// TIA Portal V16 export
// export: Created 2024-05-10T06:46:45.5884281Z, ExportSetting WithDefaults, DisplayName Totally Integrated Automation Portal, DisplayVersion V16, DisplayName TIA Portal Version Control Interface, DisplayVersion V16, DisplayName TIA Portal Openness, DisplayVersion V16, DisplayName STEP 7 Professional, DisplayVersion V16, DisplayName STEP 7 Safety, DisplayVersion V16, DisplayName WinCC Professional, DisplayVersion V16
VAR_GLOBAL   // PLC tag table "106轴控制变量表"
   轴1定位1自动 AT %M2400.0 : Bool;
   轴1定位2自动 AT %M2400.1 : Bool;
   轴1定位3自动 AT %M2400.2 : Bool;
   轴1定位4自动 AT %M2400.3 : Bool;
   轴1xx1 AT %M2400.4 : Bool;
   轴1xx2 AT %M2400.5 : Bool;
   轴1xx3 AT %M2400.6 : Bool;
   轴1xx4 AT %M2400.7 : Bool;
   轴2定位1自动 AT %M2402.0 : Bool;
   轴2定位2自动 AT %M2402.1 : Bool;
   轴2定位3自动 AT %M2402.2 : Bool;
   轴2定位4自动 AT %M2402.3 : Bool;
   轴2xx1 AT %M2402.4 : Bool;
   轴2xx2 AT %M2402.5 : Bool;
   轴2xx3 AT %M2402.6 : Bool;
   轴2xx4 AT %M2402.7 : Bool;
   轴3定位1自动 AT %M2404.0 : Bool;
   轴3定位2自动 AT %M2404.1 : Bool;
   轴3定位3自动 AT %M2404.2 : Bool;
   轴3定位4自动 AT %M2404.3 : Bool;
   轴3xx1 AT %M2404.4 : Bool;
   轴3xx2 AT %M2404.5 : Bool;
   轴3xx3 AT %M2404.6 : Bool;
   轴3xx4 AT %M2404.7 : Bool;
   轴4定位1自动 AT %M2406.0 : Bool;
   轴4定位2自动 AT %M2406.1 : Bool;
   轴4定位3自动 AT %M2406.2 : Bool;
   轴4定位4自动 AT %M2406.3 : Bool;
   轴4xx1 AT %M2406.4 : Bool;
   轴4xx2 AT %M2406.5 : Bool;
   轴4xx3 AT %M2406.6 : Bool;
   轴4xx4 AT %M2406.7 : Bool;
   轴5定位1自动 AT %M2408.0 : Bool;
   轴5定位2自动 AT %M2408.1 : Bool;
   轴5定位3自动 AT %M2408.2 : Bool;
   轴5定位4自动 AT %M2408.3 : Bool;
   轴5xx1 AT %M2408.4 : Bool;
   轴5xx2 AT %M2408.5 : Bool;
   轴5xx3 AT %M2408.6 : Bool;
   轴5xx4 AT %M2408.7 : Bool;
   轴6定位1自动 AT %M2410.0 : Bool;
   轴6定位2自动 AT %M2410.1 : Bool;
   轴6定位3自动 AT %M2410.2 : Bool;
   轴6定位4自动 AT %M2410.3 : Bool;
   轴6xx1 AT %M2410.4 : Bool;
   轴6xx2 AT %M2410.5 : Bool;
   轴6xx3 AT %M2410.6 : Bool;
   轴6xx4 AT %M2410.7 : Bool;
   轴7定位1自动 AT %M2412.0 : Bool;
   轴7定位2自动 AT %M2412.1 : Bool;
   轴7定位3自动 AT %M2412.2 : Bool;
   轴7定位4自动 AT %M2412.3 : Bool;
   轴7xx1 AT %M2412.4 : Bool;
   轴7xx2 AT %M2412.5 : Bool;
   轴7xx3 AT %M2412.6 : Bool;
   轴7xx4 AT %M2412.7 : Bool;
   轴8定位1自动 AT %M2414.0 : Bool;
   轴8定位2自动 AT %M2414.1 : Bool;
   轴8定位3自动 AT %M2414.2 : Bool;
   轴8定位4自动 AT %M2414.3 : Bool;
   轴8xx1 AT %M2414.4 : Bool;
   轴8xx2 AT %M2414.5 : Bool;
   轴8xx3 AT %M2414.6 : Bool;
   轴8xx4 AT %M2414.7 : Bool;
   轴9定位1自动 AT %M2416.0 : Bool;
   轴9定位2自动 AT %M2416.1 : Bool;
   轴9定位3自动 AT %M2416.2 : Bool;
   轴9定位4自动 AT %M2416.3 : Bool;
   轴9xx1 AT %M2416.4 : Bool;
   轴9xx2 AT %M2416.5 : Bool;
   轴9xx3 AT %M2416.6 : Bool;
   轴9xx4 AT %M2416.7 : Bool;
   轴10定位1自动 AT %M2418.0 : Bool;
   轴10定位2自动 AT %M2418.1 : Bool;
   轴10定位3自动 AT %M2418.2 : Bool;
   轴10定位4自动 AT %M2418.3 : Bool;
   轴10xx1 AT %M2418.4 : Bool;
   轴10xx2 AT %M2418.5 : Bool;
   轴10xx3 AT %M2418.6 : Bool;
   轴10xx4 AT %M2418.7 : Bool;
   轴11定位1自动 AT %M2420.0 : Bool;
   轴11定位2自动 AT %M2420.1 : Bool;
   轴11定位3自动 AT %M2420.2 : Bool;
   轴11定位4自动 AT %M2420.3 : Bool;
   轴11xx1 AT %M2420.4 : Bool;
   轴11xx2 AT %M2420.5 : Bool;
   轴11xx3 AT %M2420.6 : Bool;
   轴11xx4 AT %M2420.7 : Bool;
   轴12定位1自动 AT %M2422.0 : Bool;
   轴12定位2自动 AT %M2422.1 : Bool;
   轴12定位3自动 AT %M2422.2 : Bool;
   轴12定位4自动 AT %M2422.3 : Bool;
   轴12xx1 AT %M2422.4 : Bool;
   轴12xx2 AT %M2422.5 : Bool;
   轴12xx3 AT %M2422.6 : Bool;
   轴12xx4 AT %M2422.7 : Bool;
   轴13定位1自动 AT %M2424.0 : Bool;
   轴13定位2自动 AT %M2424.1 : Bool;
   轴13定位3自动 AT %M2424.2 : Bool;
   轴13定位4自动 AT %M2424.3 : Bool;
   轴13xx1 AT %M2424.4 : Bool;
   轴13xx2 AT %M2424.5 : Bool;
   轴13xx3 AT %M2424.6 : Bool;
   轴13xx4 AT %M2424.7 : Bool;
   轴14定位1自动 AT %M2426.0 : Bool;
   轴14定位2自动 AT %M2426.1 : Bool;
   轴14定位3自动 AT %M2426.2 : Bool;
   轴14定位4自动 AT %M2426.3 : Bool;
   轴14xx1 AT %M2426.4 : Bool;
   轴14xx2 AT %M2426.5 : Bool;
   轴14xx3 AT %M2426.6 : Bool;
   轴14xx4 AT %M2426.7 : Bool;
   轴15定位1自动 AT %M2428.0 : Bool;
   轴15定位2自动 AT %M2428.1 : Bool;
   轴15定位3自动 AT %M2428.2 : Bool;
   轴15定位4自动 AT %M2428.3 : Bool;
   轴15xx1 AT %M2428.4 : Bool;
   轴15xx2 AT %M2428.5 : Bool;
   轴15xx3 AT %M2428.6 : Bool;
   轴15xx4 AT %M2428.7 : Bool;
   轴16定位1自动 AT %M2430.0 : Bool;
   轴16定位2自动 AT %M2430.1 : Bool;
   轴16定位3自动 AT %M2430.2 : Bool;
   轴16定位4自动 AT %M2430.3 : Bool;
   轴16xx1 AT %M2430.4 : Bool;
   轴16xx2 AT %M2430.5 : Bool;
   轴16xx3 AT %M2430.6 : Bool;
   轴16xx4 AT %M2430.7 : Bool;
   XXXXXX1 AT %M2432.0 : Bool;
   轴1定位1手动 AT %M1400.0 : Bool;
   轴1定位2手动 AT %M1400.1 : Bool;
   轴1定位3手动 AT %M1400.2 : Bool;
   轴1定位4手动 AT %M1400.3 : Bool;
   轴1xx1手动 AT %M1400.4 : Bool;
   轴1xx2手动 AT %M1400.5 : Bool;
   轴1xx3手动 AT %M1400.6 : Bool;
   轴1xx4手动 AT %M1400.7 : Bool;
   轴1使能 AT %M1401.0 : Bool;
   轴1回零 AT %M1401.1 : Bool;
   "轴1点动+" AT %M1401.2 : Bool;
   "轴1点动-" AT %M1401.3 : Bool;
   轴1自由定位 AT %M1401.4 : Bool;
   轴1就绪 AT %M1401.5 : Bool;
   轴1原点 AT %M1401.6 : Bool;
   轴1到达 AT %M1401.7 : Bool;
   轴2定位1手动 AT %M1402.0 : Bool;
   轴2定位2手动 AT %M1402.1 : Bool;
   轴2定位3手动 AT %M1402.2 : Bool;
   轴2定位4手动 AT %M1402.3 : Bool;
   轴2xx1手动 AT %M1402.4 : Bool;
   轴2xx2手动 AT %M1402.5 : Bool;
   轴2xx3手动 AT %M1402.6 : Bool;
   轴2xx4手动 AT %M1402.7 : Bool;
   轴2使能 AT %M1403.0 : Bool;
   轴2回零 AT %M1403.1 : Bool;
   "轴2点动+" AT %M1403.2 : Bool;
   "轴2点动-" AT %M1403.3 : Bool;
   轴2自由定位 AT %M1403.4 : Bool;
   轴2就绪 AT %M1403.5 : Bool;
   轴2原点 AT %M1403.6 : Bool;
   轴2到达 AT %M1403.7 : Bool;
   轴3定位1手动 AT %M1404.0 : Bool;
   轴3定位2手动 AT %M1404.1 : Bool;
   轴3定位3手动 AT %M1404.2 : Bool;
   轴3定位4手动 AT %M1404.3 : Bool;
   轴3xx1手动 AT %M1404.4 : Bool;
   轴3xx2手动 AT %M1404.5 : Bool;
   轴3xx3手动 AT %M1404.6 : Bool;
   轴3xx4手动 AT %M1404.7 : Bool;
   轴3使能 AT %M1405.0 : Bool;
   轴3回零 AT %M1405.1 : Bool;
   "轴3点动+" AT %M1405.2 : Bool;
   "轴3点动-" AT %M1405.3 : Bool;
   轴3自由定位 AT %M1405.4 : Bool;
   轴3就绪 AT %M1405.5 : Bool;
   轴3原点 AT %M1405.6 : Bool;
   轴3到达 AT %M1405.7 : Bool;
   轴4定位1手动 AT %M1406.0 : Bool;
   轴4定位2手动 AT %M1406.1 : Bool;
   轴4定位3手动 AT %M1406.2 : Bool;
   轴4自由定位 AT %M1407.4 : Bool;
   轴4xx1手动 AT %M1406.4 : Bool;
   轴4xx2手动 AT %M1406.5 : Bool;
   轴4xx3手动 AT %M1406.6 : Bool;
   轴4xx4手动 AT %M1406.7 : Bool;
   轴4使能 AT %M1407.0 : Bool;
   轴4回零 AT %M1407.1 : Bool;
   "轴4点动+" AT %M1407.2 : Bool;
   "轴4点动-" AT %M1407.3 : Bool;
   轴4就绪 AT %M1407.5 : Bool;
   轴4原点 AT %M1407.6 : Bool;
   轴4到达 AT %M1407.7 : Bool;
   轴5定位1手动 AT %M1408.0 : Bool;
   轴5定位2手动 AT %M1408.1 : Bool;
   轴5定位3手动 AT %M1408.2 : Bool;
   轴5定位4手动 AT %M1408.3 : Bool;
   轴5xx1手动 AT %M1408.4 : Bool;
   轴5xx2手动 AT %M1408.5 : Bool;
   轴5xx3手动 AT %M1408.6 : Bool;
   轴5xx4手动 AT %M1408.7 : Bool;
   轴5使能 AT %M1409.0 : Bool;
   轴5回零 AT %M1409.1 : Bool;
   "轴5点动+" AT %M1409.2 : Bool;
   "轴5点动-" AT %M1409.3 : Bool;
   轴5自由定位 AT %M1409.4 : Bool;
   轴5就绪 AT %M1409.5 : Bool;
   轴5原点 AT %M1409.6 : Bool;
   轴5到达 AT %M1409.7 : Bool;
   轴6定位1手动 AT %M1410.0 : Bool;
   轴6定位2手动 AT %M1410.1 : Bool;
   轴6定位3手动 AT %M1410.2 : Bool;
   轴6定位4手动 AT %M1410.3 : Bool;
   轴6xx1手动 AT %M1410.4 : Bool;
   轴6xx2手动 AT %M1410.5 : Bool;
   轴6xx3手动 AT %M1410.6 : Bool;
   轴6xx4手动 AT %M1410.7 : Bool;
   轴6使能 AT %M1411.0 : Bool;
   轴6回零 AT %M1411.1 : Bool;
   "轴6点动+" AT %M1411.2 : Bool;
   "轴6点动-" AT %M1411.3 : Bool;
   轴6自由定位 AT %M1411.4 : Bool;
   轴6就绪 AT %M1411.5 : Bool;
   轴6原点 AT %M1411.6 : Bool;
   轴6到达 AT %M1411.7 : Bool;
   轴7定位1手动 AT %M1412.0 : Bool;
   轴7定位2手动 AT %M1412.1 : Bool;
   轴7定位3手动 AT %M1412.2 : Bool;
   轴7定位4手动 AT %M1412.3 : Bool;
   轴7xx1手动 AT %M1412.4 : Bool;
   轴7xx2手动 AT %M1412.5 : Bool;
   轴7xx3手动 AT %M1412.6 : Bool;
   轴7xx4手动 AT %M1412.7 : Bool;
   轴7使能 AT %M1413.0 : Bool;
   轴7回零 AT %M1413.1 : Bool;
   "轴7点动+" AT %M1413.2 : Bool;
   "轴7点动-" AT %M1413.3 : Bool;
   轴7自由定位 AT %M1413.4 : Bool;
   轴7就绪 AT %M1413.5 : Bool;
   轴7原点 AT %M1413.6 : Bool;
   轴7到达 AT %M1413.7 : Bool;
   轴8定位1手动 AT %M1414.0 : Bool;
   轴8定位2手动 AT %M1414.1 : Bool;
   轴8定位3手动 AT %M1414.2 : Bool;
   轴8定位4手动 AT %M1414.3 : Bool;
   轴8xx1手动 AT %M1414.4 : Bool;
   轴8xx2手动 AT %M1414.5 : Bool;
   轴8xx3手动 AT %M1414.6 : Bool;
   轴8xx4手动 AT %M1414.7 : Bool;
   轴8使能 AT %M1415.0 : Bool;
   轴8回零 AT %M1415.1 : Bool;
   "轴8点动+" AT %M1415.2 : Bool;
   "轴8点动-" AT %M1415.3 : Bool;
   轴8自由定位 AT %M1415.4 : Bool;
   轴8就绪 AT %M1415.5 : Bool;
   轴8原点 AT %M1415.6 : Bool;
   轴8到达 AT %M1415.7 : Bool;
   轴9定位1手动 AT %M1416.0 : Bool;
   轴9定位2手动 AT %M1416.1 : Bool;
   轴9定位3手动 AT %M1416.2 : Bool;
   轴9定位4手动 AT %M1416.3 : Bool;
   轴9xx1手动 AT %M1416.4 : Bool;
   轴9xx2手动 AT %M1416.5 : Bool;
   轴9xx3手动 AT %M1416.6 : Bool;
   轴9xx4手动 AT %M1416.7 : Bool;
   轴9使能 AT %M1417.0 : Bool;
   轴9回零 AT %M1417.1 : Bool;
   "轴9点动+" AT %M1417.2 : Bool;
   "轴9点动-" AT %M1417.3 : Bool;
   轴9自由定位 AT %M1417.4 : Bool;
   轴9就绪 AT %M1417.5 : Bool;
   轴9原点 AT %M1417.6 : Bool;
   轴9到达 AT %M1417.7 : Bool;
   轴10定位1手动 AT %M1418.0 : Bool;
   轴10定位2手动 AT %M1418.1 : Bool;
   轴10定位3手动 AT %M1418.2 : Bool;
   轴10定位4手动 AT %M1418.3 : Bool;
   轴10xx1手动 AT %M1418.4 : Bool;
   轴10xx2手动 AT %M1418.5 : Bool;
   轴10xx3手动 AT %M1418.6 : Bool;
   轴10xx4手动 AT %M1418.7 : Bool;
   轴10使能 AT %M1419.0 : Bool;
   轴10回零 AT %M1419.1 : Bool;
   "轴10点动+" AT %M1419.2 : Bool;
   "轴10点动-" AT %M1419.3 : Bool;
   轴10自由定位 AT %M1419.4 : Bool;
   轴10就绪 AT %M1419.5 : Bool;
   轴10原点 AT %M1419.6 : Bool;
   轴10到达 AT %M1419.7 : Bool;
   轴11定位1手动 AT %M1420.0 : Bool;
   轴11定位2手动 AT %M1420.1 : Bool;
   轴11定位3手动 AT %M1420.2 : Bool;
   轴11定位4手动 AT %M1420.3 : Bool;
   轴11xx1手动 AT %M1420.4 : Bool;
   轴11xx2手动 AT %M1420.5 : Bool;
   轴11xx3手动 AT %M1420.6 : Bool;
   轴11xx4手动 AT %M1420.7 : Bool;
   轴11使能 AT %M1421.0 : Bool;
   轴11回零 AT %M1421.1 : Bool;
   "轴11点动+" AT %M1421.2 : Bool;
   "轴11点动-" AT %M1421.3 : Bool;
   轴11自由定位 AT %M1421.4 : Bool;
   轴11就绪 AT %M1421.5 : Bool;
   轴11原点 AT %M1421.6 : Bool;
   轴11到达 AT %M1421.7 : Bool;
   轴12定位1手动 AT %M1422.0 : Bool;
   轴12定位2手动 AT %M1422.1 : Bool;
   轴12定位3手动 AT %M1422.2 : Bool;
   轴12定位4手动 AT %M1422.3 : Bool;
   轴12xx1手动 AT %M1422.4 : Bool;
   轴12xx2手动 AT %M1422.5 : Bool;
   轴12xx3手动 AT %M1422.6 : Bool;
   轴12xx4手动 AT %M1422.7 : Bool;
   轴12使能 AT %M1423.0 : Bool;
   轴12回零 AT %M1423.1 : Bool;
   "轴12点动+" AT %M1423.2 : Bool;
   "轴12点动-" AT %M1423.3 : Bool;
   轴12自由定位 AT %M1423.4 : Bool;
   轴12就绪 AT %M1423.5 : Bool;
   轴12原点 AT %M1423.6 : Bool;
   轴12到达 AT %M1423.7 : Bool;
   轴13定位1手动 AT %M1424.0 : Bool;
   轴13定位2手动 AT %M1424.1 : Bool;
   轴13定位3手动 AT %M1424.2 : Bool;
   轴13定位4手动 AT %M1424.3 : Bool;
   轴13xx1手动 AT %M1424.4 : Bool;
   轴13xx2手动 AT %M1424.5 : Bool;
   轴13xx3手动 AT %M1424.6 : Bool;
   轴13xx4手动 AT %M1424.7 : Bool;
   轴13使能 AT %M1425.0 : Bool;
   轴13回零 AT %M1425.1 : Bool;
   "轴13点动+" AT %M1425.2 : Bool;
   "轴13点动-" AT %M1425.3 : Bool;
   轴13自由定位 AT %M1425.4 : Bool;
   轴13就绪 AT %M1425.5 : Bool;
   轴13原点 AT %M1425.6 : Bool;
   轴13到达 AT %M1425.7 : Bool;
   轴14定位1手动 AT %M1426.0 : Bool;
   轴14定位2手动 AT %M1426.1 : Bool;
   轴14定位3手动 AT %M1426.2 : Bool;
   轴14定位4手动 AT %M1426.3 : Bool;
   轴14xx1手动 AT %M1426.4 : Bool;
   轴14xx2手动 AT %M1426.5 : Bool;
   轴14xx3手动 AT %M1426.6 : Bool;
   轴14xx4手动 AT %M1426.7 : Bool;
   轴14使能 AT %M1427.0 : Bool;
   轴14回零 AT %M1427.1 : Bool;
   "轴14点动+" AT %M1427.2 : Bool;
   "轴14点动-" AT %M1427.3 : Bool;
   轴14自由定位 AT %M1427.4 : Bool;
   轴14就绪 AT %M1427.5 : Bool;
   轴14原点 AT %M1427.6 : Bool;
   轴14到达 AT %M1427.7 : Bool;
   轴15定位1手动 AT %M1428.0 : Bool;
   轴15定位2手动 AT %M1428.1 : Bool;
   轴15定位3手动 AT %M1428.2 : Bool;
   轴15定位4手动 AT %M1428.3 : Bool;
   轴15xx1手动 AT %M1428.4 : Bool;
   轴15xx2手动 AT %M1428.5 : Bool;
   轴15xx3手动 AT %M1428.6 : Bool;
   轴15xx4手动 AT %M1428.7 : Bool;
   轴15使能 AT %M1429.0 : Bool;
   轴15回零 AT %M1429.1 : Bool;
   "轴15点动+" AT %M1429.2 : Bool;
   "轴15点动-" AT %M1429.3 : Bool;
   轴15自由定位 AT %M1429.4 : Bool;
   轴15就绪 AT %M1429.5 : Bool;
   轴15原点 AT %M1429.6 : Bool;
   轴15到达 AT %M1429.7 : Bool;
   轴16定位1手动 AT %M1430.0 : Bool;
   轴16定位2手动 AT %M1430.1 : Bool;
   轴16定位3手动 AT %M1430.2 : Bool;
   轴16定位4手动 AT %M1430.3 : Bool;
   轴16xx1手动 AT %M1430.4 : Bool;
   轴16xx2手动 AT %M1430.5 : Bool;
   轴16xx3手动 AT %M1430.6 : Bool;
   轴16xx4手动 AT %M1430.7 : Bool;
   轴16使能 AT %M1431.0 : Bool;
   轴16回零 AT %M1431.1 : Bool;
   "轴16点动+" AT %M1431.2 : Bool;
   "轴16点动-" AT %M1431.3 : Bool;
   轴16自由定位 AT %M1431.4 : Bool;
   轴16就绪 AT %M1431.5 : Bool;
   轴16原点 AT %M1431.6 : Bool;
   轴16到达 AT %M1431.7 : Bool;
   XXXXXX2 AT %M1432.0 : Bool;
   轴1定位1到位 AT %M3400.0 : Bool;
   轴1定位2到位 AT %M3400.1 : Bool;
   轴1定位3到位 AT %M3400.2 : Bool;
   轴1定位4到位 AT %M3400.3 : Bool;
   轴2定位1到位 AT %M3401.0 : Bool;
   轴2定位2到位 AT %M3401.1 : Bool;
   轴2定位3到位 AT %M3401.2 : Bool;
   轴2定位4到位 AT %M3401.3 : Bool;
   轴3定位1到位 AT %M3402.0 : Bool;
   轴3定位2到位 AT %M3402.1 : Bool;
   轴3定位3到位 AT %M3402.2 : Bool;
   轴3定位4到位 AT %M3402.3 : Bool;
   轴4定位1到位 AT %M3403.0 : Bool;
   轴4定位2到位 AT %M3403.1 : Bool;
   轴4定位3到位 AT %M3403.2 : Bool;
   轴4定位4到位 AT %M3403.3 : Bool;
   轴5定位1到位 AT %M3404.0 : Bool;
   轴5定位2到位 AT %M3404.1 : Bool;
   轴5定位3到位 AT %M3404.2 : Bool;
   轴5定位4到位 AT %M3404.3 : Bool;
   轴6定位1到位 AT %M3405.0 : Bool;
   轴6定位2到位 AT %M3405.1 : Bool;
   轴6定位3到位 AT %M3405.2 : Bool;
   轴6定位4到位 AT %M3405.3 : Bool;
   轴7定位1到位 AT %M3406.0 : Bool;
   轴7定位2到位 AT %M3406.1 : Bool;
   轴7定位3到位 AT %M3406.2 : Bool;
   轴7定位4到位 AT %M3406.3 : Bool;
   轴8定位1到位 AT %M3407.0 : Bool;
   轴8定位2到位 AT %M3407.1 : Bool;
   轴8定位3到位 AT %M3407.2 : Bool;
   轴8定位4到位 AT %M3407.3 : Bool;
   轴9定位1到位 AT %M3408.0 : Bool;
   轴9定位2到位 AT %M3408.1 : Bool;
   轴9定位3到位 AT %M3408.2 : Bool;
   轴9定位4到位 AT %M3408.3 : Bool;
   轴10定位1到位 AT %M3409.0 : Bool;
   轴10定位2到位 AT %M3409.1 : Bool;
   轴10定位3到位 AT %M3409.2 : Bool;
   轴10定位4到位 AT %M3409.3 : Bool;
   轴11定位1到位 AT %M3410.0 : Bool;
   轴11定位2到位 AT %M3410.1 : Bool;
   轴11定位3到位 AT %M3410.2 : Bool;
   轴11定位4到位 AT %M3410.3 : Bool;
   轴12定位1到位 AT %M3411.0 : Bool;
   轴12定位2到位 AT %M3411.1 : Bool;
   轴12定位3到位 AT %M3411.2 : Bool;
   轴12定位4到位 AT %M3411.3 : Bool;
   轴13定位1到位 AT %M3412.0 : Bool;
   轴13定位2到位 AT %M3412.1 : Bool;
   轴13定位3到位 AT %M3412.2 : Bool;
   轴13定位4到位 AT %M3412.3 : Bool;
   轴14定位1到位 AT %M3413.0 : Bool;
   轴14定位2到位 AT %M3413.1 : Bool;
   轴14定位3到位 AT %M3413.2 : Bool;
   轴14定位4到位 AT %M3413.3 : Bool;
   轴15定位1到位 AT %M3414.0 : Bool;
   轴15定位2到位 AT %M3414.1 : Bool;
   轴15定位3到位 AT %M3414.2 : Bool;
   轴15定位4到位 AT %M3414.3 : Bool;
   轴16定位1到位 AT %M3415.0 : Bool;
   轴16定位2到位 AT %M3415.1 : Bool;
   轴16定位3到位 AT %M3415.2 : Bool;
   轴16定位4到位 AT %M3415.3 : Bool;
   XXXXXX3 AT %M3416.0 : Bool;
   轴1回零高速 AT %MD1500 : DInt;
   轴1回零低速 AT %MD1504 : DInt;
   轴1点动速度 AT %MD1508 : DInt;
   轴1最高速度 AT %MD1512 : DInt;
   轴1自由定位值 AT %MD1516 : DInt;
   轴2回零高速 AT %MD1520 : DInt;
   轴2回零低速 AT %MD1524 : DInt;
   轴2点动速度 AT %MD1528 : DInt;
   轴2最高速度 AT %MD1532 : DInt;
   轴2自由定位值 AT %MD1536 : DInt;
   轴3回零高速 AT %MD1540 : DInt;
   轴3回零低速 AT %MD1544 : DInt;
   轴3点动速度 AT %MD1548 : DInt;
   轴3最高速度 AT %MD1552 : DInt;
   轴3自由定位值 AT %MD1556 : DInt;
   轴4回零高速 AT %MD1560 : DInt;
   轴4回零低速 AT %MD1564 : DInt;
   轴4点动速度 AT %MD1568 : DInt;
   轴4最高速度 AT %MD1572 : DInt;
   轴4自由定位值 AT %MD1576 : DInt;
   轴5回零高速 AT %MD1580 : DInt;
   轴5回零低速 AT %MD1584 : DInt;
   轴5点动速度 AT %MD1588 : DInt;
   轴5最高速度 AT %MD1592 : DInt;
   轴5自由定位值 AT %MD1596 : DInt;
   轴6回零高速 AT %MD1600 : DInt;
   轴6回零低速 AT %MD1604 : DInt;
   轴6点动速度 AT %MD1608 : DInt;
   轴6最高速度 AT %MD1612 : DInt;
   轴6自由定位值 AT %MD1616 : DInt;
   轴7回零高速 AT %MD1620 : DInt;
   轴7回零低速 AT %MD1624 : DInt;
   轴7点动速度 AT %MD1628 : DInt;
   轴7最高速度 AT %MD1632 : DInt;
   轴7自由定位值 AT %MD1636 : DInt;
   轴8回零高速 AT %MD1640 : DInt;
   轴8回零低速 AT %MD1644 : DInt;
   轴8点动速度 AT %MD1648 : DInt;
   轴8最高速度 AT %MD1652 : DInt;
   轴8自由定位值 AT %MD1656 : DInt;
   轴9回零高速 AT %MD1660 : DInt;
   轴9回零低速 AT %MD1664 : DInt;
   轴9点动速度 AT %MD1668 : DInt;
   轴9最高速度 AT %MD1672 : DInt;
   轴9自由定位值 AT %MD1676 : DInt;
   轴10回零高速 AT %MD1680 : DInt;
   轴10回零低速 AT %MD1684 : DInt;
   轴10点动速度 AT %MD1688 : DInt;
   轴10最高速度 AT %MD1692 : DInt;
   轴10自由定位值 AT %MD1696 : DInt;
   轴11回零高速 AT %MD1700 : DInt;
   轴11回零低速 AT %MD1704 : DInt;
   轴11点动速度 AT %MD1708 : DInt;
   轴11最高速度 AT %MD1712 : DInt;
   轴11自由定位值 AT %MD1716 : DInt;
   轴12回零高速 AT %MD1720 : DInt;
   轴12回零低速 AT %MD1724 : DInt;
   轴12点动速度 AT %MD1728 : DInt;
   轴12最高速度 AT %MD1732 : DInt;
   轴12自由定位值 AT %MD1736 : DInt;
   轴13回零高速 AT %MD1740 : DInt;
   轴13回零低速 AT %MD1744 : DInt;
   轴13点动速度 AT %MD1748 : DInt;
   轴13最高速度 AT %MD1752 : DInt;
   轴13自由定位值 AT %MD1756 : DInt;
   轴14回零高速 AT %MD1760 : DInt;
   轴14回零低速 AT %MD1764 : DInt;
   轴14点动速度 AT %MD1768 : DInt;
   轴14最高速度 AT %MD1772 : DInt;
   轴14自由定位值 AT %MD1776 : DInt;
   轴15回零高速 AT %MD1780 : DInt;
   轴15回零低速 AT %MD1784 : DInt;
   轴15点动速度 AT %MD1788 : DInt;
   轴15最高速度 AT %MD1792 : DInt;
   轴15自由定位值 AT %MD1796 : DInt;
   轴16回零高速 AT %MD1800 : DInt;
   轴16回零低速 AT %MD1804 : DInt;
   轴16点动速度 AT %MD1808 : DInt;
   轴16最高速度 AT %MD1812 : DInt;
   轴16自由定位值 AT %MD1816 : DInt;
   XXXXXX4 AT %MW1920 : Int;
   轴1位置1 AT %MD2500 : DInt;
   轴1位置2 AT %MD2504 : DInt;
   轴1位置3 AT %MD2508 : DInt;
   轴1位置4 AT %MD2512 : DInt;
   轴2位置1 AT %MD2520 : DInt;
   轴2位置2 AT %MD2524 : DInt;
   轴2位置3 AT %MD2528 : DInt;
   轴2位置4 AT %MD2532 : DInt;
   轴3位置1 AT %MD2540 : DInt;
   轴3位置2 AT %MD2544 : DInt;
   轴3位置3 AT %MD2548 : DInt;
   轴3位置4 AT %MD2552 : DInt;
   轴4位置1 AT %MD2560 : DInt;
   轴4位置2 AT %MD2564 : DInt;
   轴4位置3 AT %MD2568 : DInt;
   轴4位置4 AT %MD2572 : DInt;
   轴5位置1 AT %MD2580 : DInt;
   轴5位置2 AT %MD2584 : DInt;
   轴5位置3 AT %MD2588 : DInt;
   轴5位置4 AT %MD2592 : DInt;
   轴6位置1 AT %MD2600 : DInt;
   轴6位置2 AT %MD2604 : DInt;
   轴6位置3 AT %MD2608 : DInt;
   轴6位置4 AT %MD2612 : DInt;
   轴7位置1 AT %MD2620 : DInt;
   轴7位置2 AT %MD2624 : DInt;
   轴7位置3 AT %MD2628 : DInt;
   轴7位置4 AT %MD2632 : DInt;
   轴8位置1 AT %MD2640 : DInt;
   轴8位置2 AT %MD2644 : DInt;
   轴8位置3 AT %MD2648 : DInt;
   轴8位置4 AT %MD2652 : DInt;
   轴9位置1 AT %MD2660 : DInt;
   轴9位置2 AT %MD2664 : DInt;
   轴9位置3 AT %MD2668 : DInt;
   轴9位置4 AT %MD2672 : DInt;
   轴10位置1 AT %MD2680 : DInt;
   轴10位置2 AT %MD2684 : DInt;
   轴10位置3 AT %MD2688 : DInt;
   轴10位置4 AT %MD2692 : DInt;
   轴11位置1 AT %MD2700 : DInt;
   轴11位置2 AT %MD2704 : DInt;
   轴11位置3 AT %MD2708 : DInt;
   轴11位置4 AT %MD2712 : DInt;
   轴12位置1 AT %MD2720 : DInt;
   轴12位置2 AT %MD2724 : DInt;
   轴12位置3 AT %MD2728 : DInt;
   轴12位置4 AT %MD2732 : DInt;
   轴13位置1 AT %MD2740 : DInt;
   轴13位置2 AT %MD2744 : DInt;
   轴13位置3 AT %MD2748 : DInt;
   轴13位置4 AT %MD2752 : DInt;
   轴14位置1 AT %MD2760 : DInt;
   轴14位置2 AT %MD2764 : DInt;
   轴14位置3 AT %MD2768 : DInt;
   轴14位置4 AT %MD2772 : DInt;
   轴15位置1 AT %MD2780 : DInt;
   轴15位置2 AT %MD2784 : DInt;
   轴15位置3 AT %MD2788 : DInt;
   轴15位置4 AT %MD2792 : DInt;
   轴16位置1 AT %MD2800 : DInt;
   轴16位置2 AT %MD2804 : DInt;
   轴16位置3 AT %MD2808 : DInt;
   轴16位置4 AT %MD2812 : DInt;
   XXXXXX5 AT %MW2820 : Int;
   轴1速度1 AT %MW3500 : Int;
   轴1速度2 AT %MW3504 : Int;
   轴1速度3 AT %MW3508 : Int;
   轴1速度4 AT %MW3512 : Int;
   轴2速度1 AT %MW3520 : Int;
   轴2速度2 AT %MW3524 : Int;
   轴2速度3 AT %MW3528 : Int;
   轴2速度4 AT %MW3532 : Int;
   轴3速度1 AT %MW3540 : Int;
   轴3速度2 AT %MW3544 : Int;
   轴3速度3 AT %MW3548 : Int;
   轴3速度4 AT %MW3552 : Int;
   轴4速度1 AT %MW3560 : Int;
   轴4速度2 AT %MW3564 : Int;
   轴4速度3 AT %MW3568 : Int;
   轴4速度4 AT %MW3572 : Int;
   轴5速度1 AT %MW3580 : Int;
   轴5速度2 AT %MW3584 : Int;
   轴5速度3 AT %MW3588 : Int;
   轴5速度4 AT %MW3592 : Int;
   轴6速度1 AT %MW3600 : Int;
   轴6速度2 AT %MW3604 : Int;
   轴6速度3 AT %MW3608 : Int;
   轴6速度4 AT %MW3612 : Int;
   轴7速度1 AT %MW3620 : Int;
   轴7速度2 AT %MW3624 : Int;
   轴7速度3 AT %MW3628 : Int;
   轴7速度4 AT %MW3632 : Int;
   轴8速度1 AT %MW3640 : Int;
   轴8速度2 AT %MW3644 : Int;
   轴8速度3 AT %MW3648 : Int;
   轴8速度4 AT %MW3652 : Int;
   轴9速度1 AT %MW3660 : Int;
   轴9速度2 AT %MW3664 : Int;
   轴9速度3 AT %MW3668 : Int;
   轴9速度4 AT %MW3672 : Int;
   轴10速度1 AT %MW3680 : Int;
   轴10速度2 AT %MW3684 : Int;
   轴10速度3 AT %MW3688 : Int;
   轴10速度4 AT %MW3692 : Int;
   轴11速度1 AT %MW3700 : Int;
   轴11速度2 AT %MW3704 : Int;
   轴11速度3 AT %MW3708 : Int;
   轴11速度4 AT %MW3712 : Int;
   轴12速度1 AT %MW3720 : Int;
   轴12速度2 AT %MW3724 : Int;
   轴12速度3 AT %MW3728 : Int;
   轴12速度4 AT %MW3732 : Int;
   轴13速度1 AT %MW3740 : Int;
   轴13速度2 AT %MW3744 : Int;
   轴13速度3 AT %MW3748 : Int;
   轴13速度4 AT %MW3752 : Int;
   轴14速度1 AT %MW3760 : Int;
   轴14速度2 AT %MW3764 : Int;
   轴14速度3 AT %MW3768 : Int;
   轴14速度4 AT %MW3772 : Int;
   轴15速度1 AT %MW3780 : Int;
   轴15速度2 AT %MW3784 : Int;
   轴15速度3 AT %MW3788 : Int;
   轴15速度4 AT %MW3792 : Int;
   轴16速度1 AT %MW3800 : Int;
   轴16速度2 AT %MW3804 : Int;
   轴16速度3 AT %MW3808 : Int;
   轴16速度4 AT %MW3812 : Int;
   XXXXXX6 AT %MW3820 : Int;
   轴01目标位置 AT %MD4500 : DInt;
   轴02目标位置 AT %MD4504 : DInt;
   轴03目标位置 AT %MD4508 : DInt;
   轴04目标位置 AT %MD4512 : DInt;
   轴05目标位置 AT %MD4516 : DInt;
   轴06目标位置 AT %MD4520 : DInt;
   轴07目标位置 AT %MD4524 : DInt;
   轴08目标位置 AT %MD4528 : DInt;
   轴09目标位置 AT %MD4532 : DInt;
   轴10目标位置 AT %MD4536 : DInt;
   轴11目标位置 AT %MD4540 : DInt;
   轴12目标位置 AT %MD4544 : DInt;
   轴13目标位置 AT %MD4548 : DInt;
   轴14目标位置 AT %MD4552 : DInt;
   轴15目标位置 AT %MD4556 : DInt;
   轴16目标位置 AT %MD4560 : DInt;
   XXXXXX7 AT %MD4564 : DInt;
   轴01目标速度 AT %MD4600 : DInt;
   轴02目标速度 AT %MD4604 : DInt;
   轴03目标速度 AT %MD4608 : DInt;
   轴04目标速度 AT %MD4612 : DInt;
   轴05目标速度 AT %MD4616 : DInt;
   轴06目标速度 AT %MD4620 : DInt;
   轴07目标速度 AT %MD4624 : DInt;
   轴08目标速度 AT %MD4628 : DInt;
   轴09目标速度 AT %MD4632 : DInt;
   轴10目标速度 AT %MD4636 : DInt;
   轴11目标速度 AT %MD4640 : DInt;
   轴12目标速度 AT %MD4644 : DInt;
   轴13目标速度 AT %MD4648 : DInt;
   轴14目标速度 AT %MD4652 : DInt;
   轴15目标速度 AT %MD4656 : DInt;
   轴16目标速度 AT %MD4660 : DInt;
   XXXXXX8 AT %MD4664 : DInt;
   轴01当前位置 AT %MD4700 : DInt;
   轴02当前位置 AT %MD4704 : DInt;
   轴03当前位置 AT %MD4708 : DInt;
   轴04当前位置 AT %MD4712 : DInt;
   轴05当前位置 AT %MD4716 : DInt;
   轴06当前位置 AT %MD4720 : DInt;
   轴07当前位置 AT %MD4724 : DInt;
   轴08当前位置 AT %MD4728 : DInt;
   轴09当前位置 AT %MD4732 : DInt;
   轴10当前位置 AT %MD4736 : DInt;
   轴11当前位置 AT %MD4740 : DInt;
   轴12当前位置 AT %MD4744 : DInt;
   轴13当前位置 AT %MD4748 : DInt;
   轴14当前位置 AT %MD4752 : DInt;
   轴15当前位置 AT %MD4756 : DInt;
   轴16当前位置 AT %MD4760 : DInt;
   XXXXXX9 AT %MD4764 : DInt;
   轴01当前速度 AT %MD4800 : DInt;
   轴02当前速度 AT %MD4804 : DInt;
   轴03当前速度 AT %MD4808 : DInt;
   轴04当前速度 AT %MD4812 : DInt;
   轴05当前速度 AT %MD4816 : DInt;
   轴06当前速度 AT %MD4820 : DInt;
   轴07当前速度 AT %MD4824 : DInt;
   轴08当前速度 AT %MD4828 : DInt;
   轴09当前速度 AT %MD4832 : DInt;
   轴10当前速度 AT %MD4836 : DInt;
   轴11当前速度 AT %MD4840 : DInt;
   轴12当前速度 AT %MD4844 : DInt;
   轴13当前速度 AT %MD4848 : DInt;
   轴14当前速度 AT %MD4852 : DInt;
   轴15当前速度 AT %MD4856 : DInt;
   轴16当前速度 AT %MD4860 : DInt;
   XXXXXX10 AT %MD4864 : DInt;
   轴1报警码 AT %MW4900 : Word;
   轴2报警码 AT %MW4901 : Word;
   轴3报警码 AT %MW4902 : Word;
   轴4报警码 AT %MW4903 : Word;
   轴5报警码 AT %MW4904 : Word;
   轴6报警码 AT %MW4905 : Word;
   轴7报警码 AT %MW4906 : Word;
   轴8报警码 AT %MW4907 : Word;
   轴9报警码 AT %MW4908 : Word;
   轴10报警码 AT %MW4909 : Word;
   轴11报警码 AT %MW4910 : Word;
   轴12报警码 AT %MW4911 : Word;
   轴13报警码 AT %MW4912 : Word;
   轴14报警码 AT %MW4913 : Word;
   轴15报警码 AT %MW4914 : Word;
   轴16报警码 AT %MW4915 : Word;
   XXXXXX11 AT %MW4916 : Word;
   轴1错误码 AT %MW4920 : Word;
   轴2错误码 AT %MW4921 : Word;
   轴3错误码 AT %MW4922 : Word;
   轴4错误码 AT %MW4923 : Word;
   轴5错误码 AT %MW4924 : Word;
   轴6错误码 AT %MW4925 : Word;
   轴7错误码 AT %MW4926 : Word;
   轴8错误码 AT %MW4927 : Word;
   轴9错误码 AT %MW4928 : Word;
   轴10错误码 AT %MW4929 : Word;
   轴11错误码 AT %MW4930 : Word;
   轴12错误码 AT %MW4931 : Word;
   轴13错误码 AT %MW4932 : Word;
   轴14错误码 AT %MW4933 : Word;
   轴15错误码 AT %MW4934 : Word;
   轴16错误码 AT %MW4935 : Word;
END_VAR
